FUNCTION_BLOCK Axis
VAR_INPUT
END_VAR
VAR_OUTPUT
END_VAR
VAR
	i:INT;
END_VAR

// NETWORK 1

END_FUNCTION_BLOCK

(* stored: Version 1.1.0.1, ProductVersion 3.1.4024.4
   POU Axis: Id {9a29a284-b343-4c08-8559-93ac28bec8ca}, SpecialFunc None *)
